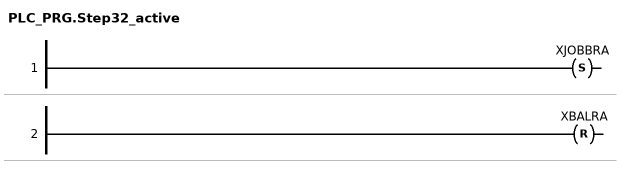
// NETWORK 1
XJOBBRA S= TRUE;

// NETWORK 2
XBALRA R= TRUE;
END_ACTION

ACTION Step33_active:
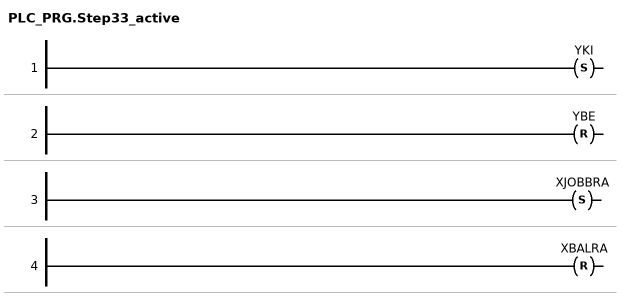
// NETWORK 1
YKI S= TRUE;

// NETWORK 2
YBE R= TRUE;

// NETWORK 3
XJOBBRA S= TRUE;

// NETWORK 4
XBALRA R= TRUE;
END_ACTION

ACTION Step36_active:
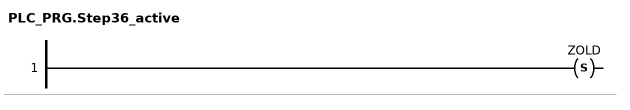
// NETWORK 1
ZOLD S= TRUE;
END_ACTION

END_PROGRAM
